Staubli VAL3: OnF2.pgx

program OnF2()
  local num l_ni
  local bool l_bRes
  local string l_sItem
begin
  //
  switch nPage
    //新建产品
    case 0
      call setPrd(sList,l_sItem)
      if l_sItem!=""
        if sPrd[nSelected]!=""
          nSelected=nSelected+1
          insert(sPrd[nSelected])
          insert(sProductList[nSelected])
        endIf
        sPrd[nSelected]=l_sItem
        sProductList[nSelected]=""
      endIf
    break
    //插入路径
    case 1
      call InsertPath()
    break
  endSwitch
  bUserRefresh=bListRefresh=true
end
